SUBAPPLICATION Uebung_056 (* DigitalInput_I1-_I4 auf DigitalOutput_Q1-_Q4 *)
  (* Standard: 61499-2 *)
  (* Version 1.0, 2023-10-23, franz *)
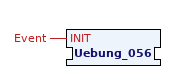
  EVENT_INPUT
    INIT;
  END_EVENT
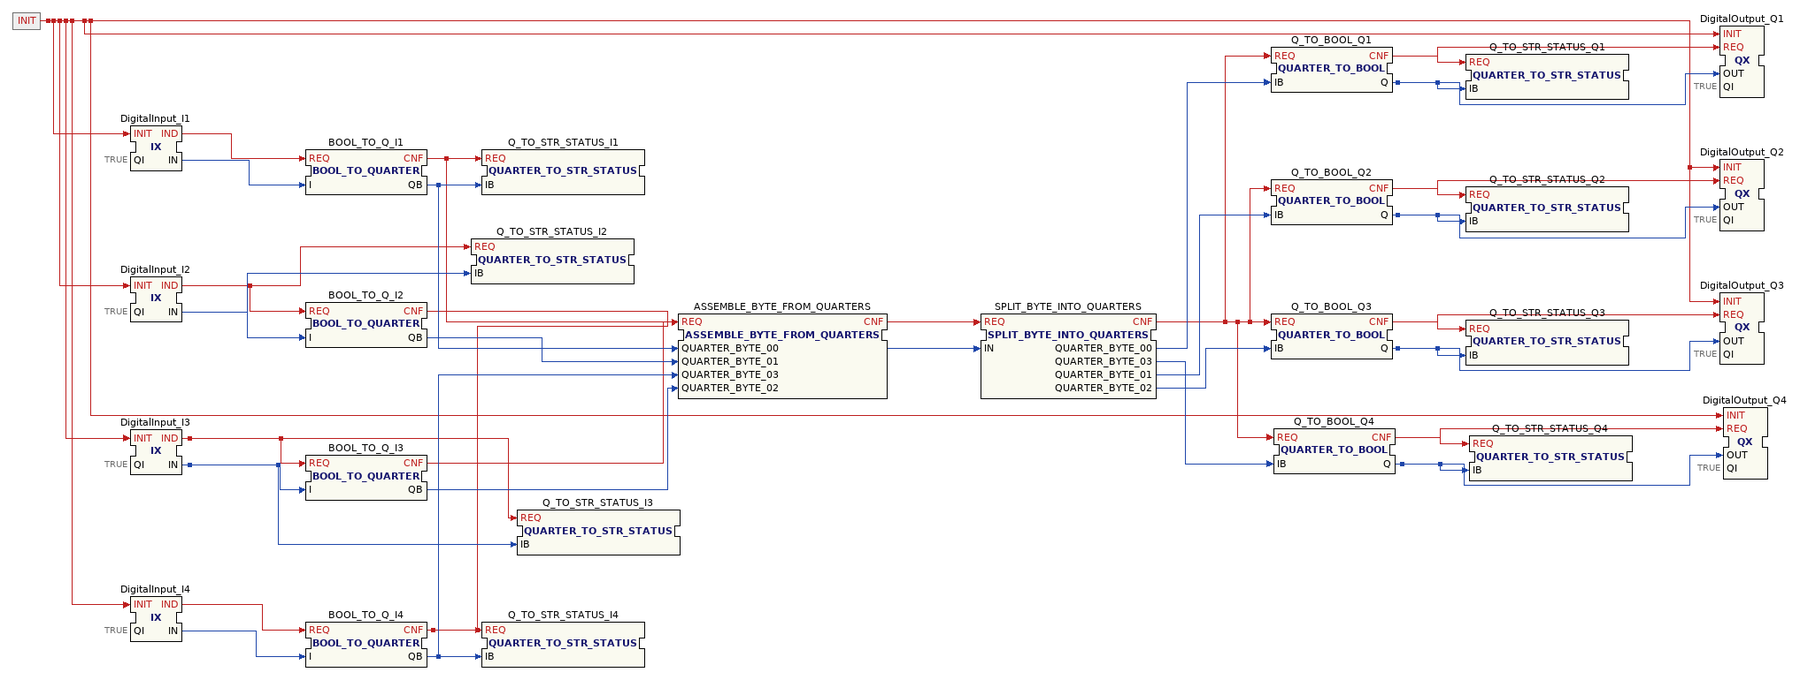
  FBS
    DigitalInput_I1 : IX(QI := TRUE);
    ASSEMBLE_BYTE_FROM_QUARTERS : ASSEMBLE_BYTE_FROM_QUARTERS;
    DigitalInput_I2 : IX(QI := TRUE);
    DigitalInput_I3 : IX(QI := TRUE);
    DigitalInput_I4 : IX(QI := TRUE);
    DigitalOutput_Q2 : QX(QI := TRUE);
    DigitalOutput_Q3 : QX(QI := TRUE);
    SPLIT_BYTE_INTO_QUARTERS : SPLIT_BYTE_INTO_QUARTERS;
    DigitalOutput_Q1 : QX(QI := TRUE);
    DigitalOutput_Q4 : QX(QI := TRUE);
    Q_TO_BOOL_Q1 : QUARTER_TO_BOOL;
    Q_TO_BOOL_Q4 : QUARTER_TO_BOOL;
    Q_TO_BOOL_Q2 : QUARTER_TO_BOOL;
    Q_TO_BOOL_Q3 : QUARTER_TO_BOOL;
    Q_TO_STR_STATUS_Q3 : QUARTER_TO_STR_STATUS;
    Q_TO_STR_STATUS_Q1 : QUARTER_TO_STR_STATUS;
    Q_TO_STR_STATUS_I3 : QUARTER_TO_STR_STATUS;
    Q_TO_STR_STATUS_I1 : QUARTER_TO_STR_STATUS;
    Q_TO_STR_STATUS_I4 : QUARTER_TO_STR_STATUS;
    Q_TO_STR_STATUS_Q4 : QUARTER_TO_STR_STATUS;
    Q_TO_STR_STATUS_Q2 : QUARTER_TO_STR_STATUS;
    Q_TO_STR_STATUS_I2 : QUARTER_TO_STR_STATUS;
    BOOL_TO_Q_I1 : BOOL_TO_QUARTER;
    BOOL_TO_Q_I2 : BOOL_TO_QUARTER;
    BOOL_TO_Q_I4 : BOOL_TO_QUARTER;
    BOOL_TO_Q_I3 : BOOL_TO_QUARTER;
  END_FBS
  EVENT_CONNECTIONS
    INIT TO DigitalInput_I1.INIT;
    INIT TO DigitalInput_I2.INIT;
    INIT TO DigitalInput_I3.INIT;
    INIT TO DigitalInput_I4.INIT;
    ASSEMBLE_BYTE_FROM_QUARTERS.CNF TO SPLIT_BYTE_INTO_QUARTERS.REQ;
    INIT TO DigitalOutput_Q1.INIT;
    INIT TO DigitalOutput_Q4.INIT;
    INIT TO DigitalOutput_Q3.INIT;
    INIT TO DigitalOutput_Q2.INIT;
    SPLIT_BYTE_INTO_QUARTERS.CNF TO Q_TO_BOOL_Q1.REQ;
    Q_TO_BOOL_Q1.CNF TO DigitalOutput_Q1.REQ;
    SPLIT_BYTE_INTO_QUARTERS.CNF TO Q_TO_BOOL_Q4.REQ;
    Q_TO_BOOL_Q4.CNF TO DigitalOutput_Q4.REQ;
    SPLIT_BYTE_INTO_QUARTERS.CNF TO Q_TO_BOOL_Q2.REQ;
    Q_TO_BOOL_Q2.CNF TO DigitalOutput_Q2.REQ;
    SPLIT_BYTE_INTO_QUARTERS.CNF TO Q_TO_BOOL_Q3.REQ;
    Q_TO_BOOL_Q3.CNF TO DigitalOutput_Q3.REQ;
    Q_TO_BOOL_Q3.CNF TO Q_TO_STR_STATUS_Q3.REQ;
    Q_TO_BOOL_Q1.CNF TO Q_TO_STR_STATUS_Q1.REQ;
    DigitalInput_I3.IND TO Q_TO_STR_STATUS_I3.REQ;
    Q_TO_BOOL_Q4.CNF TO Q_TO_STR_STATUS_Q4.REQ;
    Q_TO_BOOL_Q2.CNF TO Q_TO_STR_STATUS_Q2.REQ;
    DigitalInput_I2.IND TO Q_TO_STR_STATUS_I2.REQ;
    DigitalInput_I1.IND TO BOOL_TO_Q_I1.REQ;
    BOOL_TO_Q_I1.CNF TO ASSEMBLE_BYTE_FROM_QUARTERS.REQ;
    BOOL_TO_Q_I1.CNF TO Q_TO_STR_STATUS_I1.REQ;
    DigitalInput_I2.IND TO BOOL_TO_Q_I2.REQ;
    BOOL_TO_Q_I2.CNF TO ASSEMBLE_BYTE_FROM_QUARTERS.REQ;
    DigitalInput_I4.IND TO BOOL_TO_Q_I4.REQ;
    BOOL_TO_Q_I4.CNF TO ASSEMBLE_BYTE_FROM_QUARTERS.REQ;
    BOOL_TO_Q_I4.CNF TO Q_TO_STR_STATUS_I4.REQ;
    DigitalInput_I3.IND TO BOOL_TO_Q_I3.REQ;
    BOOL_TO_Q_I3.CNF TO ASSEMBLE_BYTE_FROM_QUARTERS.REQ;
  END_CONNECTIONS
  DATA_CONNECTIONS
    Q_TO_BOOL_Q1.Q TO DigitalOutput_Q1.OUT;
    Q_TO_BOOL_Q4.Q TO DigitalOutput_Q4.OUT;
    Q_TO_BOOL_Q2.Q TO DigitalOutput_Q2.OUT;
    Q_TO_BOOL_Q3.Q TO DigitalOutput_Q3.OUT;
    Q_TO_BOOL_Q3.Q TO Q_TO_STR_STATUS_Q3.IB;
    Q_TO_BOOL_Q1.Q TO Q_TO_STR_STATUS_Q1.IB;
    DigitalInput_I3.IN TO Q_TO_STR_STATUS_I3.IB;
    Q_TO_BOOL_Q4.Q TO Q_TO_STR_STATUS_Q4.IB;
    Q_TO_BOOL_Q2.Q TO Q_TO_STR_STATUS_Q2.IB;
    DigitalInput_I2.IN TO Q_TO_STR_STATUS_I2.IB;
    DigitalInput_I1.IN TO BOOL_TO_Q_I1.I;
    BOOL_TO_Q_I1.QB TO Q_TO_STR_STATUS_I1.IB;
    DigitalInput_I2.IN TO BOOL_TO_Q_I2.I;
    DigitalInput_I4.IN TO BOOL_TO_Q_I4.I;
    BOOL_TO_Q_I4.QB TO Q_TO_STR_STATUS_I4.IB;
    DigitalInput_I3.IN TO BOOL_TO_Q_I3.I;
    ASSEMBLE_BYTE_FROM_QUARTERS. TO SPLIT_BYTE_INTO_QUARTERS.IN;
    SPLIT_BYTE_INTO_QUARTERS.QUARTER_BYTE_00 TO Q_TO_BOOL_Q1.IB;
    SPLIT_BYTE_INTO_QUARTERS.QUARTER_BYTE_03 TO Q_TO_BOOL_Q4.IB;
    SPLIT_BYTE_INTO_QUARTERS.QUARTER_BYTE_01 TO Q_TO_BOOL_Q2.IB;
    SPLIT_BYTE_INTO_QUARTERS.QUARTER_BYTE_02 TO Q_TO_BOOL_Q3.IB;
    BOOL_TO_Q_I1.QB TO ASSEMBLE_BYTE_FROM_QUARTERS.QUARTER_BYTE_00;
    BOOL_TO_Q_I2.QB TO ASSEMBLE_BYTE_FROM_QUARTERS.QUARTER_BYTE_01;
    BOOL_TO_Q_I4.QB TO ASSEMBLE_BYTE_FROM_QUARTERS.QUARTER_BYTE_03;
    BOOL_TO_Q_I3.QB TO ASSEMBLE_BYTE_FROM_QUARTERS.QUARTER_BYTE_02;
  END_CONNECTIONS
END_SUBAPPLICATION
